FUNCTION_BLOCK FB_Axis
VAR_INPUT
END_VAR
VAR_OUTPUT
END_VAR
VAR
	axis	: AXIS_REF;
	mcPower	: MC_Power;
	mcMove	: MC_MoveAbsolute;
	mcReset	: MC_Reset;
	fbAlarm	: FB_TcAlarm;
	
	_error	: BOOL;
	_errorId	: UDINT;
END_VAR

METHOD AbsMove : BOOL
VAR_INPUT
	Execute	: BOOL;
	Position	: LREAL;
	Velocity	: LREAL;
END_VAR
VAR_INST
	nState	: INT;
	rTrig	: R_TRIG;
END_VAR
AbsMove := FALSE;

rTrig(Clk := Execute);
IF rTrig.Q THEN
	nState := 10;
	mcMove(Axis := Axis, Execute := FALSE);
END_IF

IF NOT Execute THEN
	nState := 0;
END_IF

CASE nState OF
	10: // move
		mcMove.Position := Position;
		mcMove.Velocity := Velocity;
		mcMove.Execute := TRUE;
		IF McMove.Done THEN
			nState := 20;
			mcMove.Execute := FALSE;
		END_IF
		IF mcMove.Error THEN
			_error := TRUE;
			_errorId := mcMove.ErrorID;
			fbAlarm.ipArguments.Clear().AddUDInt(_errorId);
			fbAlarm.Raise(0);
			mcMove.Execute := FALSE;
			nState := 20;
		END_IF
		mcMove(Axis := Axis);
	20: // done state
		AbsMove := TRUE;
END_CASE
END_METHOD

METHOD Disable : BOOL
VAR_INPUT
END_VAR
Axis.ReadStatus();
Disable := NOT mcPower.Status;
mcPower(Axis := Axis, Enable := FALSE);
END_METHOD

METHOD Enable : BOOL
VAR_INPUT
END_VAR
axis.ReadStatus();
Enable := mcPower.Status AND axis.Status.Operational;
mcPower(axis := axis, enable := TRUE, Enable_Positive := TRUE, Enable_Negative := TRUE);
END_METHOD

PROPERTY Error : BOOL
GET
Error := Axis.NcToPlc.ErrorCode <> 0 OR _error;
END_GET
END_PROPERTY

METHOD FB_init : BOOL
VAR_INPUT
	bInitRetains : BOOL; // if TRUE, the retain variables are initialized (warm start / cold start)
	bInCopyCode : BOOL;  // if TRUE, the instance afterwards gets moved into the copy code (online change)
END_VAR
IF fbAlarm.EqualsToEventEntryEx(stOther := TC_EVENTS.SlitterEvents.EjectorAxisError) THEN
	fbAlarm.CreateEx(TC_EVENTS.SlitterEvents.EjectorAxisError, FALSE, 0);
	fbAlarm.ipArguments.Clear();
END_IF
END_METHOD

PROPERTY IsEnabled : BOOL
GET
Axis.ReadStatus();
IsEnabled := mcPower.Status AND Axis.Status.Operational;
END_GET
END_PROPERTY

METHOD Reset : BOOL
VAR_INPUT
	Execute : BOOL;
END_VAR
VAR_INST
	nState	: INT;
	rTrig	: R_TRIG;
END_VAR
Reset := FALSE;
rTrig(CLK := Execute);
IF rTrig.Q THEN
	mcMove(Axis := Axis, Execute := FALSE);
	mcReset(Axis := Axis, Execute := FALSE);
	_error := FALSE;
	_errorId := 0;
	nState := 10;
END_IF
IF NOT Execute THEN
	nState := 0;
END_IF
CASE nState OF
	10: // reset the system
		IF fbAlarm.bRaised THEN
			fbAlarm.Clear(0, FALSE);
		END_IF
		mcReset.Execute := TRUE;
		IF mcReset.Done THEN
			mcReset.Execute := FALSE;
			nState := 20;
		END_IF
		IF mcReset.Error THEN
			_error := TRUE;
			_errorId := mcReset.ErrorID;
			fbAlarm.ipArguments.Clear().AddUDInt(_errorId);
			fbAlarm.Raise(0);
			nState := 20;
		END_IF
		mcReset(Axis := Axis);
	20: // done state
		Reset := TRUE;
END_CASE
END_METHOD

END_FUNCTION_BLOCK

(* stored: Version 1.1.0.1, ProductVersion 3.1.4024.9
   POU FB_Axis: Id {bc000919-1c04-4722-abe2-41d5cc74783b}, SpecialFunc None
   Method AbsMove: Id {c2f4b0ca-b88e-4fc8-9492-63069fb84dce}
   Method Disable: Id {eeabe391-6cd3-4d46-a266-e62f3d58dd8b}
   Method Enable: Id {32dab039-f63c-4cef-a370-2213ac51175c}
   Property Error: Id {7e1079a6-5dbd-4dad-86f5-5f117f277c72}
   Get Get: Id {a5dc245c-87aa-4c5f-940d-b1bdc5cc5441}
   Method FB_init: Id {23fc91f8-4e71-4631-ad5d-1b88e434a24a}
   Property IsEnabled: Id {60a7f699-9173-473c-a2cb-1674d9ee927f}
   Get Get: Id {d4c7f1fe-6918-46c6-96a1-06914821be66}
   Method Reset: Id {a90c0f7c-f40b-41f5-b12f-9195c5c5b06f} *)
